Universal Robots URScript: motion_capture.script

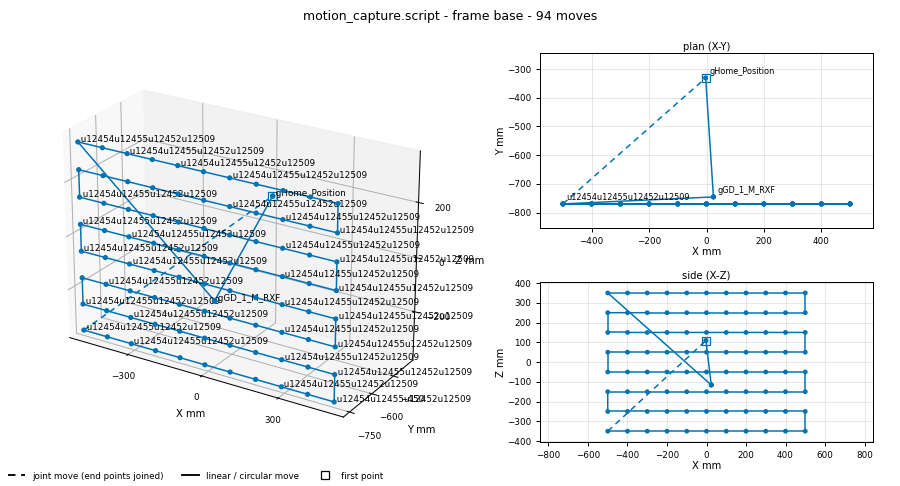
[picture p0: tool path of motion_capture.script in frame base, 94 of 94 moves have a stored position in this frame; points joined in program order, loops and branches not executed]
def motion_capture():
  global _hidden_verificationVariable=0
  set_standard_analog_input_domain(0, 1)
  set_standard_analog_input_domain(1, 1)
  set_tool_analog_input_domain(0, 1)
  set_tool_analog_input_domain(1, 1)
  set_analog_outputdomain(0, 0)
  set_analog_outputdomain(1, 0)
  set_input_actions_to_default()
  set_runstate_gp_boolean_output_to_value(0, 3)
  set_tcp(p[0.0,0.08,0.42,0.0,0.0,0.0])
  set_target_payload(0.100000, [0.135000, 0.000000, 0.225000], [10.000000, 10.000000, 10.000000, 0.000000, 0.000000, 0.000000])
  set_gravity([0.0, 0.0, 9.82])
  set_tool_communication(False, 115200, 0, 1, 1.5, 3.5)
  set_tool_output_mode(0)
  set_tool_digital_output_mode(0, 1)
  set_tool_digital_output_mode(1, 1)
  set_tool_voltage(0)
  set_safety_mode_transition_hardness(1)
  global DistPillar=0.26672
  global CandCnt=1
  global ReCaptZ=0.05
  global port=3000
  global socket_timeout=120
  global host="192.168.1.2"
  global is_popup=False
  global pBucket=[p[0.79266, 0.38712, 0.34284, 0, 0, -1.59403], p[-0.74859, -0.57465, 0.33542, 0, 0, 1.57589], p[0, 0, 0, 0, 0, 0]]
  global CaptStepZ=0.085
  global CaptIndex=[0, 0, 0]
  global pBucketM=p[-0.76064, -0.49997, 0.35503, 0, 0, 1.57135]
  global socket_name="vt"
  global rovi_err=0
  global SubPrgResult=100
  global CurrPos=p[-0.00509, -0.40914, 0.52153, -0.02622, -3.13819, -0.00861]
  global CurrPos_p=p[-0.00512, -0.32683, 0.10197, -0.02622, -3.13819, -0.00861]
  global ForceStartZ=0.4
  global CutOffZ=0.08
  global Sub3100_ZMax=0.74
  global ForceStartX=-0.90368
  global Sub3100_aRot=0.2
  global Sub3100_d=0.3
  global Sub3100_Option=3
  global Sub3100_a=0.2
  global Sub3100_XdV=0.1
  global Sub3100_XdRot=8
  global ZoneDistTh=0.05
  global BucketWidth=0.95
  global ZoneBucketGap=0
  global ZoneHomeX=0.2
  global UnloadZ=0.06
  global CaptPos=p[0.47573, -0.4259, 0.04497, 3.14138, 0.03448, 0.00005]
  global BucketUpperPos=p[0.47573, -0.4259, 0.04497, 3.14138, 0.03448, 0.00005]
  global Sub3100_GPII18=3
  global Zone6ThX=0.1
  global Zone6ThY=0.05
  global pCV=p[0.0013, 0.00002, 0.00241, 0.00218, 0.00027, 0.00056]
  global CaptRowNo=0
  global CrankDepthFull=0.025
  global CrankDepth=0.42751
  global Y1=[1, 266.72156, 0, 0]
  global Y2=p[0.01216, -0.30795, 0.04758, -0.01683, 0.01631, -1.59125]
  global EvacRadiusTh=0.3
  global EvacXTh=[-0.5, 0.5]
  global EvacYTh=[-0.8, 1]
  global EvacZTh=[-0.1, 0.1]
  global WorkPosNo=1
  global Zone1ZTh=0.1
  global ReCaptNo=0
  global DistPillarBak=0.26672
  global CaptIndexWk=0
  global PoseSub=p[-0.02953, -0.26506, -0.34451, -0.05387, -0.00646, 0.16446]
  global PoseAdd=p[-0.83785, 0.22711, 0.71052, 2.06849, 2.21352, 0.02519]
  global RZTh=15
  global pBucketC=p[0.45, -0.8, 0.35, 0, 0, 3.1415]
  global ReCaptZWk=0
  global CheckMST=2
  global RZSub=9.42295
  global DistPillarCOTh=0.16
  global DistPillarAPTh=0.25
  global CutOffZAdd=0.03
  global CutOffZDef=0.08
  global Y8=0
  global BKWidth_Value=[950, 986, 0]
  global BKWidth_Name="/prepro/bucket_width"
  global Bucket=p[0.32604,0.49174,0.0,-1.882900624652718E-5,2.8304179127934987E-5,-1.593185305749222]
  global BucketM=p[0.32604,0.49174,0.0,2.2353980716304163E-16,-3.5868426080024975E-16,-1.5931853071795856]
  global CV=p[0.0,0.0,0.0,0.0,0.0,0.0]
  global CaptPoint_C=p[-0.335,-0.024,0.4,-2.196299060524223,-2.2462891909035143,-5.664484063487096E-5]
  global CaptPoint_C2=p[0.32796661698047924,-0.010768520544682924,0.01931625281283378,2.2288103429550152,-2.213636886217198,8.598462540813273E-5]
  global CaptPoint_L=p[-0.335,-0.246,0.4,2.1515798175986935,2.2007172931471577,-0.09388261158531223]
  global CaptPoint_L2=p[0.327894307417917,-0.010799940826224014,0.01928712668893995,2.087717047309385,-2.0736781215133306,0.27365839887453103]
  global CaptPoint_R=p[-0.335,0.246,0.4,-2.1517289105627166,-2.2005994980169152,-0.09391633243318627]
  global CaptPoint_R2=p[0.327926308680866,-0.010795166414457658,0.019300245403843563,-2.1186306375223185,2.1040550557443427,0.22023197678473694]
  global Capt_1BK_L=p[-0.395,-0.47,0.35,-2.1961210242572884,-2.2463362846055,-2.908274762447041E-4]
  global Capt_1BK_R=p[-0.395,0.51,0.35,2.196067754706757,2.246288285862388,2.8411291050601595E-5]
  global Capt_1BK_pos1=p[-0.4218793038724447,-0.003154429464978058,0.2915499891144615,-2.1963422029204875,-2.2438663520270015,-0.02197160668673838]
  global Capt_1BK_pos2=p[-0.42187829024618434,-0.0031710253373066375,0.29156503858953065,-2.196324918349679,-2.2439040699490773,-0.021928444416953782]
  global Capt_2BK_L=p[0.42186661528427194,0.4254738068040517,0.35042275762909847,2.239156309475874,-2.1837044610999294,0.002643817066643282]
  global Capt_2BK_R=p[0.4218208572756906,-0.5427676723257963,0.350372239919558,2.2392697861179327,-2.183553596194912,0.002410470905346486]
  global Capt_2BK_pos1=p[0.42193501458435656,0.004742683868356356,0.35045865974037793,2.2391012408536453,-2.1839704655717003,0.002677867056024068]
  global Capt_2BK_pos2=p[0.421903984494575,0.004707988774967922,0.35045218900915065,2.239114367170047,-2.183895515396197,0.002684056681074047]
  global Capt_CV_M=p[-0.04794223960540197,-0.559868557160475,0.1086937653706071,-0.022464429848058916,-3.141454018347238,4.0166993855964835E-4]
  global Capt_GD_M=p[-0.004053197679954899,-0.25261725691632436,-0.01970497430780127,0.0332779454553888,-3.140179196376707,-0.0034093680964018282]
  global HomePointL=p[-0.36789,-0.5117344641471838,0.78,-0.6278857271586024,3.0680899128661667,-8.649957362498864E-4]
  global Master_pos=p[-0.003,-0.27,0.109,-0.02099899522131702,-3.141447277644474,4.6083856157132165E-4]
  global Master_posL=p[-0.003,-0.27,0.109,0.02094395102393583,3.0543261909900803,-5.235987755386035E-4]
  global Master_posR=p[-0.003,-0.27,0.109,-0.019810987664379186,-3.054193931591229,4.952746915529204E-4]
  global PickPos=p[0.10830682331105715,-1.3709505888096256,-0.18404188875951455,-0.00622194000158997,2.880236948927292,-0.00383636509397631]
  global Solve=p[-0.00368,-0.0021000000000000003,0.25739999999999996,0.0,0.0,0.0]
  global TCP3100TL=p[0.0,0.06,0.535,1.8939999999999997,0.0,0.0]
  global TEST=p[0.1,0.0,0.2,0.0,0.0,0.0]
  global UF=p[0.0,0.0,0.0,0.0,0.0,0.0]
  global g1CV_posL1=p[0.05028133628211688,-0.4526481033729615,0.1221845548632916,-2.213335080948508,-2.1937561336067057,-0.3280056759040735]
  global g1CV_posR1=p[0.03743870476062511,-0.53119407812668,0.11301901343688614,2.073418671558482,2.153257467049566,0.11656306439039889]
  global g1GD_pos1=p[0.14857012745627257,-0.6379982996093139,0.2691918735517042,2.214277610229479,2.228493098198348,-1.6896832945346036E-4]
  global g1GD_pos2=p[0.028634297882679793,-0.4702313285867709,0.450031657325677,2.214319081558633,2.2285182736309666,-1.5473710223511705E-5]
  global g1GD_pos3=p[-0.1945307709581842,-0.42906455111749103,0.45,-2.685709191057467,-1.6297557787554324,7.112239955701245E-5]
  global g1GD_pos4=p[-0.25628841794770224,-0.020630481098425146,0.45,2.148716725221303,2.2918109407224354,-1.3854918368741778E-5]
  global g1GD_pos5=p[-0.714365317693782,-0.022971007293656684,0.45,-2.1476725881724037,-2.292771958266831,6.311233907547867E-5]
  global g1GD_posL1=p[-0.08276848269606216,-0.3996147100031649,0.1488453551331823,2.286527078917204,1.8420745504477611,0.33698451773695576]
  global g1GD_posL2=p[-0.3253977027403738,-0.3024804624281039,0.16332814085945146,2.72312820760317,0.9631021078169197,0.32447452035226126]
  global g1GD_posL3=p[-0.6791033397183219,0.06787475590683856,0.16337212788108813,2.1383125299263996,2.086116032377724,0.4536080263755059]
  global g1GD_posR1=p[-0.09893370538053747,-0.4999608954567234,0.14329885217724153,2.43311852414254,1.4238397520832589,0.08559216753941556]
  global g1GD_posR2=p[-0.3729565201882258,-0.3752983669473301,0.143299052800563,2.6951655216297596,0.8130506811102118,-0.02387549506099888]
  global g1GD_posR3=p[-0.7385929502572233,-0.029472684480355026,0.1499650660949685,2.0484522752014467,1.9493695704119496,0.18368227556562683]
  global g2CV_posL1=p[0.3409386496330911,-0.4656338066361442,0.1250074988128972,2.209372209162659,2.1945371304665926,0.3160714960040194]
  global g2CV_posR1=p[0.3400736278759575,-0.531334269888987,0.1183415684753657,2.07314649492589,2.1532617466521136,0.11638666128062146]
  global g2GD_pos1=p[0.2541383831722086,-0.6774928758666339,0.18519960582577166,-2.0375719953016755,-2.3889847960447277,-0.0020926217702447064]
  global g2GD_pos2=p[0.2548303032832998,-0.4395886120507379,0.2986557393825452,-1.8691601740155521,-2.5210138137905886,-0.00387894312889377]
  global g2GD_pos3=p[0.3379879014596998,-0.06467509721500111,0.3,-0.13681955358471554,3.138134920213652,0.0052602971824959885]
  global g2GD_pos4=p[0.31412137931928874,0.14047894136547145,0.3,1.0726627132331576,-2.952135651121033,-0.005044331815994264]
  global g2GD_pos5=p[0.596826867485263,0.012800854207951809,0.3,-2.250960447020382,2.191482163995288,-8.62049956035814E-5]
  global gCV_11_M=p[0.2895856132087369,-0.9700402997477822,-0.03048660701646616,2.1152349881492576,2.082454134650371,0.2907202126305862]
  global gCV_12_M=p[0.3399735651774522,-0.9701152791174454,-0.030398240983259495,2.1151309943729695,2.082422893849917,0.2905107745619789]
  global gCV_13_M=p[0.3677028242565019,-0.8912043588518235,0.06406475497489328,2.0725171273330782,1.9964853271438565,0.36457536397978224]
  global gCV_1_M=p[0.26662,-0.9702099878169796,-0.021959001781271192,-2.212353529315613,-2.2195544467592487,0.0323655800559973]
  global gCV_2_M=p[0.26859807289598814,-0.9702702137427199,0.029436000792852024,-2.212446744366122,-2.219572570655569,0.03244046687031327]
  global gCV_3_M=p[0.29099390607376485,-0.6570558385379063,0.0722153583041818,1.9884242634571576,2.2321538498123994,0.15249643504377583]
  global gCV_pos5=p[0.3400172856834047,-0.9722754606605235,-0.18287928563575456,2.073394561413637,2.1531827558666565,0.11639000988241816]
  global gGD_1_LM=p[0.02419,-0.7289500000000001,-0.11494,-0.010169347158913017,2.870767181856166,0.2884627079222753]
  global gGD_1_LM_RX=p[0.05369459866460638,-0.7259829268100212,-0.22783950231933825,0.3045827799067659,1.9676452376021116,-2.225919618395937]
  global gGD_1_LM_RXF=p[0.02413503458160308,-0.74534,-0.11578000000000001,0.2411332216392182,1.7407173006243832,-2.3674279033231747]
  global gGD_1_M=p[0.023469999999999998,-0.72661,-0.11456000000000001,-0.029570847824802682,-3.12419917405015,-0.3106340785404749]
  global gGD_1_M_RX=p[0.023057660296999655,-0.7236214973426132,-0.23125683282505294,-0.014877844076808725,-2.067340942848176,2.343588104915257]
  global gGD_1_M_RXF=p[0.02415523713330076,-0.7453200000000001,-0.11578426509069895,-0.012477314995716382,-1.853515977408631,2.515027308648709]
  global gGD_1_RM=p[0.023629999999999998,-0.72653,-0.11331000000000001,-0.06253229749015264,-2.8808212567082414,-0.28238046714011755]
  global gGD_1_RM_RX=p[-0.005088870384171898,-0.7236679006721032,-0.22637303238730694,0.2593876111855818,-1.9494145656951658,2.2163695295960366]
  global gGD_1_RM_RXF=p[0.024158234647744328,-0.74536,-0.11577,0.21548497967238725,-1.726437707763004,2.3373117534316665]
  global gGD_2_LM=p[0.02467,-0.67055,-0.11509,-0.010179461791212513,2.870955921048522,0.2878734195391217]
  global gGD_2_LM_RX=p[0.05420311073735988,-0.6676020823088724,-0.22799649297520497,0.30453821192036695,1.967284185886619,-2.2263172758170806]
  global gGD_2_LM_RXF=p[0.02518,-0.6822999999999999,-0.11982,0.24121310672797797,1.7407223643292684,-2.3672997334921986]
  global gGD_2_M=p[0.02389,-0.6721900000000001,-0.11456000000000001,-0.029666521928107308,-3.1243201149134068,-0.3098990972493868]
  global gGD_2_M_RX=p[0.023451397096722927,-0.6694131949440525,-0.2312112380080017,-0.014956274784115499,-2.0665404158707275,2.344308336230428]
  global gGD_2_M_RXF=p[0.02469,-0.68228,-0.11781,-0.012625584579695818,-1.8536977166603092,2.514979910589354]
  global gGD_2_RM=p[0.02429,-0.66916,-0.11353,-0.06253008389277029,-2.880917079483223,-0.28230802316028863]
  global gGD_2_RM_RX=p[-0.004446905642647561,-0.6662749600062835,-0.22659916730049184,0.25917451838034067,-1.9493834256574814,2.2163998591438716]
  global gGD_2_RM_RXF=p[0.02418,-0.68221,-0.11985,0.21545635593876583,-1.7267658137434814,2.337110041109278]
  global gGD_3_LM=p[0.024149999999999998,-0.63442,-0.00372,-0.010168641563882792,2.8709293839329573,0.28786844960240987]
  global gGD_3_LM_RX=p[0.05363363651684515,-0.6315154925298007,-0.11660858214565634,0.3044658366193896,1.9671814668034862,-2.2263956155853166]
  global gGD_3_LM_RXF=p[0.02387752228160463,-0.5964211774687285,-0.05792315514989682,0.2704410553277331,1.9481847980902196,-2.214876983085744]
  global gGD_3_M=p[0.023940000000000003,-0.63613,-0.00522,-0.029962916255114207,-3.1241595671421933,-0.3100480455299553]
  global gGD_3_M_RX=p[0.023480543069899083,-0.6332104768802226,-0.1219058093136538,-0.014942206094503903,-2.066644773324154,2.3438407418712903]
  global gGD_3_M_RXF=p[0.02383447419609676,-0.5964085561522618,-0.0579509198373786,-0.014600929068906539,-2.066655165579624,2.3438719244209403]
  global gGD_3_RM=p[0.02428,-0.6347200000000001,-0.00846,-0.0624152449577923,-2.8809080008278345,-0.2823877130468296]
  global gGD_3_RM_RX=p[-0.004516944470436435,-0.6317425605459723,-0.12157603214553458,0.2593921862362061,-1.9496410574300858,2.2162312511396824]
  global gGD_3_RM_RXF=p[0.023773322279514588,-0.5964087734876792,-0.05795139315103717,0.24060086319727583,-1.933030903056379,2.187075285864524]
  global gGD_4_LM=p[-0.12534109989305553,-0.6345452257364079,-0.003660409912739915,-0.010209507081901941,2.87092276677584,0.2878514545752189]
  global gGD_4_RM=p[0.1741356102640685,-0.6348673415405857,-0.008407071546374267,-0.06250935255312234,-2.8810578033032743,-0.28204363282303685]
  global gHome_Position=p[-0.0028799999999999997,-0.33081,0.1087,-0.02099958342773921,-3.141491282453575,3.986162810876369E-4]
  global gTAIHI_pos1=p[0.034435296708333146,-0.2890869270984411,0.28697762766096685,-0.9517096680276043,2.9907327255336362,-0.006242657270483182]
  global gTAIHI_pos2=p[0.46041690381401934,0.09562026346103787,0.3409455343940188,-2.575428180750575,1.7504967205574518,-0.009370784990557466]
  global gTAIHI_pos3=p[0.4777514786587304,0.10855417509450788,0.25667938190447326,-3.115092130529677,-0.059113053813058626,0.017060902648732133]
  global gTAIHI_pos4=p[0.47773948064032057,0.10853581553326999,-0.15133852019421468,-3.1151611852917296,-0.05914313994407087,0.017149581050184888]
  global gTAIHI_pos5=p[0.30588450070104545,0.17870028478253597,-0.38750721344025674,-3.115302721311487,-0.05927431563397507,0.01725874757592571]
  rtde_set_watchdog("speed_slider_mask", 10.0, "ignore")
  # begin: URCap Installation Node
  #   Source: Ethernet/IP I/O Monitor URCap, 1.0.0,
  #   Type: Ethernet/IP I/O Monitor
  conn = rpc_factory("xmlrpc", "http://127.0.0.1:" + to_str(61101) + "/RPC2")

  def show_monitor():
    return conn.eip_monitor.show()
  end
  # end: URCap Installation Node
  step_count_397ec1da_4bf5_4cd9_852d_7e56d1a44991 = 0.0
  thread Step_Counter_Thread_d30562aa_f9e6_4b1c_b905_026c51a4cdd0():
    while (True):
      step_count_397ec1da_4bf5_4cd9_852d_7e56d1a44991 = step_count_397ec1da_4bf5_4cd9_852d_7e56d1a44991 + 1.0
      sync()
    end
  end
  run Step_Counter_Thread_d30562aa_f9e6_4b1c_b905_026c51a4cdd0()
  global u12454u12455u12452u12509u12452u12531u12488_1_p=p[-.500000000000, -.769756443525, .350000000000, .026412316980, 3.122703155576, .190069130431]
  global u12454u12455u12452u12509u12452u12531u12488_1_q=[-1.9114113979977487, -2.2618906676528763, -0.4591602097308458, -2.1103464893291033, 1.5382040123912875, -0.3218736006056453]
  global u12454u12455u12452u12509u12452u12531u12488_2_p=p[-.400000000000, -.769779294180, .350000000000, .026483300731, 3.122677399875, .189931430077]
  global u12454u12455u12452u12509u12452u12531u12488_2_q=[-1.8171775039295675, -2.133570399697568, -0.6739164307743053, -2.0258656041570973, 1.5500367362507816, -0.22781589719288586]
  global u12454u12455u12452u12509u12452u12531u12488_3_p=p[-.300000000000, -.769789509042, .350000000000, .026503166818, 3.122680364614, .190021042089]
  global u12454u12455u12452u12509u12452u12531u12488_3_q=[-1.716165423221513, -2.0483178045096206, -0.8067403790800718, -1.9793255819153632, 1.5626303580459329, -0.12725853176687707]
  global u12454u12455u12452u12509u12452u12531u12488_4_p=p[-.200000000000, -.769710320339, .350000000000, .026644809517, 3.122684897999, .190163528053]
  global u12454u12455u12452u12509u12452u12531u12488_4_q=[-1.6099254452403873, -1.9903140904082264, -0.8928752732962089, -1.9509751362852477, 1.5758064426187728, -0.021545386634477026]
  global u12454u12455u12452u12509u12452u12531u12488_5_p=p[-.100000000000, -.769748949148, .350000000000, .026539604733, 3.122630476655, .190199683938]
  global u12454u12455u12452u12509u12452u12531u12488_5_q=[-1.5005112395057907, -1.9556374381444463, -0.9429912511335443, -1.9338143920604765, 1.5892342589142574, 0.08710325076008775]
  global u12454u12455u12452u12509u12452u12531u12488_6_p=p[-.000000000000, -.769753039159, .350000000000, .026417422847, 3.122605840141, .190062143068]
  global u12454u12455u12452u12509u12452u12531u12488_6_q=[-1.3903873476760396, -1.9425809473745055, -0.9620710317474312, -1.924501091481389, 1.6023466178665648, 0.19644588241672967]
  global u12454u12455u12452u12509u12452u12531u12488_7_p=p[.100000000000, -.769697827339, .350000000000, .026676373995, 3.122609886009, .190250248267]
  global u12454u12455u12452u12509u12452u12531u12488_7_q=[-1.2822308148508128, -1.951096029905166, -0.9510725611357058, -1.9225876310592298, 1.6147201968064984, 0.3041064480521222]
  global u12454u12455u12452u12509u12452u12531u12488_8_p=p[.200000000000, -.769720790847, .350000000000, .026556961083, 3.122644596660, .190093490077]
  global u12454u12455u12452u12509u12452u12531u12488_8_q=[-1.17843186168205, -1.9812086634530637, -0.9092976431058046, -1.9286067868835772, 1.6258983197269878, 0.4072497591845611]
  global u12454u12455u12452u12509u12452u12531u12488_9_p=p[.300000000000, -.769733702676, .350000000000, .026566917094, 3.122644604456, .190111967042]
  global u12454u12455u12452u12509u12452u12531u12488_9_q=[-1.0809947819676138, -2.0340650931016366, -0.832913028063154, -1.9458910758426562, 1.6357754765791155, 0.5041839537901349]
  global u12454u12455u12452u12509u12452u12531u12488_10_p=p[.400000000000, -.769744499214, .350000000000, .026575326306, 3.122733131353, .190132184073]
  global u12454u12455u12452u12509u12452u12531u12488_10_q=[-0.991056047875758, -2.112822831401303, -0.7130015422450269, -1.9804884405124454, 1.6441329192153846, 0.5936653453753264]
  global u12454u12455u12452u12509u12452u12531u12488_11_p=p[.500000000000, -.769782793267, .350000000000, .026508483411, 3.122675353931, .190004333780]
  global u12454u12455u12452u12509u12452u12531u12488_11_q=[-0.9092045285356001, -2.2282728608507227, -0.5245252474117779, -2.0467514170930947, 1.6511301529893736, 0.674987056963054]
  global u12454u12455u12452u12509u12452u12531u12488_12_p=p[.500000000000, -.769760900368, .250000000000, .026528118536, 3.122708730810, .190029220965]
  global u12454u12455u12452u12509u12452u12531u12488_12_q=[-0.91001526414599, -2.1575818481165623, -0.8234281729531467, -1.8186342475237138, 1.6514532038321557, 0.674277213721763]
  global u12454u12455u12452u12509u12452u12531u12488_13_p=p[.400000000000, -.769733463067, .250000000000, .026514979020, 3.122645894238, .190244682604]
  global u12454u12455u12452u12509u12452u12531u12488_13_q=[-0.9917864872644486, -2.066558737990783, -0.9638838946787551, -1.775946946298058, 1.6445187709217466, 0.5928948733369976]
  global u12454u12455u12452u12509u12452u12531u12488_14_p=p[.300000000000, -.769779850713, .250000000000, .026486137196, 3.122687044148, .190087115632]
  global u12454u12455u12452u12509u12452u12531u12488_14_q=[-1.0815959341128414, -1.9988992643907082, -1.0626874450643164, -1.7513322373267535, 1.6359840099262097, 0.5034994136646239]
  global u12454u12455u12452u12509u12452u12531u12488_15_p=p[.200000000000, -.769781810740, .250000000000, .026484014283, 3.122705057460, .190154645546]
  global u12454u12455u12452u12509u12452u12531u12488_15_q=[-1.178993777620991, -1.9517406172159042, -1.1285374498245746, -1.7389315215400138, 1.6260890541146251, 0.4065892996566263]
  global u12454u12455u12452u12509u12452u12531u12488_16_p=p[.100000000000, -.769767054232, .250000000000, .026526291040, 3.122613308500, .190027323171]
  global u12454u12455u12452u12509u12452u12531u12488_16_q=[-1.2827714411646953, -1.9240889198247118, -1.165721384028017, -1.7348376877857614, 1.614912560975787, 0.3034134866458757]
  global u12454u12455u12452u12509u12452u12531u12488_17_p=p[-.000000000000, -.769774212018, .250000000000, .026548873992, 3.122655101521, .190254700093]
  global u12454u12455u12452u12509u12452u12531u12488_17_q=[-1.3909214332126858, -1.9163049894413131, -1.1754366000499896, -1.737561855870414, 1.6025377303774226, 0.19593182526004416]
  global u12454u12455u12452u12509u12452u12531u12488_18_p=p[-.100000000000, -.769761106494, .250000000000, .026526373802, 3.122686049502, .190157333824]
  global u12454u12455u12452u12509u12452u12531u12488_18_q=[-1.501031671994486, -1.9279015874596954, -1.1588712635165734, -1.7456586341412317, 1.5894077694755506, 0.08651688314535733]
  global u12454u12455u12452u12509u12452u12531u12488_19_p=p[-.200000000000, -.769774136564, .250000000000, .026456934430, 3.122604840588, .190033566826]
  global u12454u12455u12452u12509u12452u12531u12488_19_q=[-1.6105390632010685, -1.9591661196706518, -1.1149754495250734, -1.759952863358695, 1.5761181644969744, -0.02233440855401625]
  global u12454u12455u12452u12509u12452u12531u12488_20_p=p[-.300000000000, -.769781720580, .250000000000, .026577890837, 3.122652970758, .190179047147]
  global u12454u12455u12452u12509u12452u12531u12488_20_q=[-1.7167999596103485, -2.010364020103964, -1.0415152543063009, -1.7826055876402425, 1.5628826553775266, -0.12787467040920664]
  global u12454u12455u12452u12509u12452u12531u12488_21_p=p[-.400000000000, -.769744400680, .250004230661, .026455713576, 3.122633726963, .190216871674]
  global u12454u12455u12452u12509u12452u12531u12488_21_q=[-1.8178876271517623, -2.0823453079114493, -0.9341277490262669, -1.8170533568045393, 1.5502952050585215, -0.22852714499667925]
  global u12454u12455u12452u12509u12452u12531u12488_22_p=p[-.500000000000, -.769752806148, .249977272123, .026544126851, 3.122621458039, .190284973089]
  global u12454u12455u12452u12509u12452u12531u12488_22_q=[-1.912334332224173, -2.179253324474807, -0.7817836665202043, -1.870495209636136, 1.53856375120108, -0.32259002476777]
  global u12454u12455u12452u12509u12452u12531u12488_23_p=p[-.500000000000, -.769728484770, .150000000000, .026393123076, 3.122651774268, .190178886745]
  global u12454u12455u12452u12509u12452u12531u12488_23_q=[-1.9128442312041365, -2.1609661241967473, -0.987071729191296, -1.683405002467147, 1.538744683268341, -0.32326048625640524]
  global u12454u12455u12452u12509u12452u12531u12488_24_p=p[-.400000000000, -.769776260329, .150000000000, .026496921071, 3.122616212816, .190058872149]
  global u12454u12455u12452u12509u12452u12531u12488_24_q=[-1.8183484767892821, -2.0756758619090068, -1.119625076860153, -1.638125740464143, 1.5504998869009539, -0.2290611172505086]
  global u12454u12455u12452u12509u12452u12531u12488_25_p=p[-.300000000000, -.769742523564, .149972007931, .026671481565, 3.122589595262, .190100603900]
  global u12454u12455u12452u12509u12452u12531u12488_25_q=[-1.7172499604707783, -2.0100622561114037, -1.217213616444221, -1.6071690471086697, 1.5630915763257234, -0.1283793186395803]
  global u12454u12455u12452u12509u12452u12531u12488_26_p=p[-.200000000000, -.769780338502, .149978041748, .026528023660, 3.122636425681, .190070149226]
  global u12454u12455u12452u12509u12452u12531u12488_26_q=[-1.610892382818097, -1.9627414022092786, -1.2852160392852294, -1.5861622342848385, 1.5762157500238576, -0.02275843600603178]
  global u12454u12455u12452u12509u12452u12531u12488_27_p=p[-.100000000000, -.769745881180, .149995549479, .026451519491, 3.122618883192, .190101837112]
  global u12454u12455u12452u12509u12452u12531u12488_27_q=[-1.5014170801735727, -1.9334650534417097, -1.3264985118771904, -1.5724417136414282, 1.5895919353511783, 0.08595968623292746]
  global u12454u12455u12452u12509u12452u12531u12488_28_p=p[.000000000000, -.769794456996, .149992141995, .026554396761, 3.122606353239, .190010846636]
  global u12454u12455u12452u12509u12452u12531u12488_28_q=[-1.3912924404706617, -1.9226155501285076, -1.3421332945507913, -1.5644092481035372, 1.6026905136881453, 0.19544350978913963]
  global u12454u12455u12452u12509u12452u12531u12488_29_p=p[.100000000000, -.769806987713, .149985740336, .026560443917, 3.122586219799, .189931438497]
  global u12454u12455u12452u12509u12452u12531u12488_29_q=[-1.2831438437635398, -1.9302091184868697, -1.332632629894107, -1.5617624067960563, 1.6150494824601616, 0.3029425526560603]
  global u12454u12455u12452u12509u12452u12531u12488_30_p=p[.200000000000, -.769814423607, .150010855459, .026516643396, 3.122584097137, .189982361164]
  global u12454u12455u12452u12509u12452u12531u12488_30_q=[-1.1794180535327925, -1.956237208193265, -1.2974749489939068, -1.5653811410892091, 1.6262953338083186, 0.40606816526849876]
  global u12454u12455u12452u12509u12452u12531u12488_31_p=p[.300000000000, -.769831553064, .150060942487, .026545222581, 3.122662417995, .189866103692]
  global u12454u12455u12452u12509u12452u12531u12488_31_q=[-1.0819925902355525, -2.0002866059266946, -1.2357744304054723, -1.576750564863108, 1.6360955536829191, 0.5030348882059403]
  global u12454u12455u12452u12509u12452u12531u12488_32_p=p[.400000000000, -.769795781366, .150028602698, .026503365861, 3.122587531329, .189968750155]
  global u12454u12455u12452u12509u12452u12531u12488_32_q=[-0.9922270738397705, -2.0624181412994282, -1.1453333100908685, -1.5984937767840375, 1.6446469758576996, 0.5923566878529133]
  global u12454u12455u12452u12509u12452u12531u12488_33_p=p[.500000000000, -.769793999499, .150020314544, .026447218837, 3.122575290255, .189986171446]
  global u12454u12455u12452u12509u12452u12531u12488_33_q=[-0.9105654759643107, -2.1436878918100923, -1.0211433188916939, -1.634766430642408, 1.6517313132940015, 0.6736049555830492]
  global u12454u12455u12452u12509u12452u12531u12488_34_p=p[.500000000000, -.769779861568, .050000000000, .026542041208, 3.122557555389, .190062616528]
  global u12454u12455u12452u12509u12452u12531u12488_34_q=[-0.9108895793250085, -2.1632011203124684, -1.1662261267105478, -1.4702404330490406, 1.6518725992844814, 0.6731792662005232]
  global u12454u12455u12452u12509u12452u12531u12488_35_p=p[.400000000000, -.769760513107, .050000000000, .026549866540, 3.122587439777, .190000613354]
  global u12454u12455u12452u12509u12452u12531u12488_35_q=[-0.9924845968610327, -2.0881935330063115, -1.2831795311436416, -1.4349224479921512, 1.6447338235902051, 0.5919582930454563]
  global u12454u12455u12452u12509u12452u12531u12488_36_p=p[.300000000000, -.769793437396, .050000000000, .026367160197, 3.122672293278, .190001319070]
  global u12454u12455u12452u12509u12452u12531u12488_36_q=[-1.0822201887748832, -2.0301660421005394, -1.3699155602403739, -1.4128452711626203, 1.636174279208616, 0.5025162468030526]
  global u12454u12455u12452u12509u12452u12531u12488_37_p=p[.200000000000, -.769726213919, .050000000000, .026627232633, 3.122697997976, .190137353324]
  global u12454u12455u12452u12509u12452u12531u12488_37_q=[-1.1795709628866948, -1.9885443352899195, -1.4298833078132702, -1.4008180335198368, 1.6262735945297104, 0.40581240128416063]
  global u12454u12455u12452u12509u12452u12531u12488_38_p=p[.100000000000, -.769733672147, .050000000000, .026554565165, 3.122685196493, .190232809370]
  global u12454u12455u12452u12509u12452u12531u12488_38_q=[-1.283303317577559, -1.963915417659761, -1.4641828291134331, -1.3967363080991797, 1.6150349457186142, 0.3026044310190157]
  global u12454u12455u12452u12509u12452u12531u12488_39_p=p[.000000000000, -.769785322216, .050000000000, .026510503638, 3.122723125005, .190004512455]
  global u12454u12455u12452u12509u12452u12531u12488_39_q=[-1.3914339238266074, -1.9565180079824351, -1.4737422544074672, -1.3989224808881673, 1.6026155458683435, 0.1951072590510945]
  global u12454u12455u12452u12509u12452u12531u12488_40_p=p[-.100000000000, -.769765413659, .050000000000, .026427054269, 3.122646229983, .190092806256]
  global u12454u12455u12452u12509u12452u12531u12488_40_q=[-1.5016202252969766, -1.9667091354205404, -1.458514209701086, -1.407185734712944, 1.5896005709127916, 0.0855699677390378]
  global u12454u12455u12452u12509u12452u12531u12488_41_p=p[-.200000000000, -.769712657217, .050000000000, .026669437619, 3.122668765801, .190172396507]
  global u12454u12455u12452u12509u12452u12531u12488_41_q=[-1.6111137968452418, -1.9941576858132901, -1.4184742805621404, -1.4215535025581794, 1.5762220127117197, -0.023059579298967847]
  global u12454u12455u12452u12509u12452u12531u12488_42_p=p[-.300000000000, -.769708675215, .050000000000, .026592329375, 3.122688586472, .190100650432]
  global u12454u12455u12452u12509u12452u12531u12488_42_q=[-1.717446082348145, -2.038485220608205, -1.3528387367862003, -1.443102243336619, 1.563050842151673, -0.1287922067915055]
  global u12454u12455u12452u12509u12452u12531u12488_43_p=p[-.400000000000, -.769723587764, .050000000000, .026548087776, 3.122655882932, .190070701895]
  global u12454u12455u12452u12509u12452u12531u12488_43_q=[-1.8186227366851835, -2.099509098658128, -1.259828810329843, -1.4740780696228883, 1.5505307857911361, -0.22946732186074925]
  global u12454u12455u12452u12509u12452u12531u12488_44_p=p[-.500000000000, -.769745444991, .050000000000, .026448305973, 3.122671770036, .190070038317]
  global u12454u12455u12452u12509u12452u12531u12488_44_q=[-1.913168549752596, -2.1777485306121296, -1.1359749765764775, -1.5176355928160845, 1.5388491761007717, -0.3237064384801265]
  global u12454u12455u12452u12509u12452u12531u12488_45_p=p[-.500000000000, -.769748044989, -.050000000000, .026459265213, 3.122632683617, .190122460314]
  global u12454u12455u12452u12509u12452u12531u12488_45_q=[-1.9133780773117284, -2.2211331388335616, -1.2450197950729933, -1.3652385838548202, 1.5388943999966873, -0.32413817674840395]
  global u12454u12455u12452u12509u12452u12531u12488_46_p=p[-.400000000000, -.769739650303, -.050000000000, .026524363418, 3.122756240847, .190055765096]
  global u12454u12455u12452u12509u12452u12531u12488_46_q=[-1.8187371277192126, -2.1486524407136685, -1.3647457810366612, -1.3199753277104946, 1.5504419407841503, -0.22982482924301184]
  global u12454u12455u12452u12509u12452u12531u12488_47_p=p[-.300000000000, -.769776202108, -.050000000000, .026395617042, 3.122681115272, .190056900613]
  global u12454u12455u12452u12509u12452u12531u12488_47_q=[-1.7175787153903785, -2.091961769853695, -1.4555700035182593, -1.286866813305382, 1.5630389047729167, -0.1292835164360282]
  global u12454u12455u12452u12509u12452u12531u12488_48_p=p[-.200000000000, -.769746729862, -.050000000000, .026524482261, 3.122666596847, .190157077818]
  global u12454u12455u12452u12509u12452u12531u12488_48_q=[-1.6112382773031273, -2.050586009680634, -1.5203481415147833, -1.263245226402418, 1.5761868010532227, -0.023506832417726997]
  global u12454u12455u12452u12509u12452u12531u12488_49_p=p[-.100000000000, -.769781536209, -.050000000000, .026509312290, 3.122634166369, .189996544206]
  global u12454u12455u12452u12509u12452u12531u12488_49_q=[-1.5017608226441368, -2.0249283672268668, -1.5600934719950121, -1.2473325509067834, 1.589570965909667, 0.08525364952997627]
  global u12454u12455u12452u12509u12452u12531u12488_50_p=p[-.000000000000, -.769750846669, -.050000000000, .026510672437, 3.122715317755, .189959048159]
  global u12454u12455u12452u12509u12452u12531u12488_50_q=[-1.3915520266447254, -2.0154486486529937, -1.5752093407577448, -1.2385065815255096, 1.6025755644109516, 0.19476181077474664]
  global u12454u12455u12452u12509u12452u12531u12488_51_p=p[.100000000000, -.769758377488, -.050000000000, .026415226178, 3.122608928546, .189993842825]
  global u12454u12455u12452u12509u12452u12531u12488_51_q=[-1.2834508712456465, -2.022498172237963, -1.5655654952664868, -1.2366210119909358, 1.6150294159800644, 0.30214056754365615]
  global u12454u12455u12452u12509u12452u12531u12488_52_p=p[.200000000000, -.769741232078, -.050000000000, .026477631813, 3.122639493213, .190040124831]
  global u12454u12455u12452u12509u12452u12531u12488_52_q=[-1.1797194426026554, -2.0457471515932006, -1.5312483524744307, -1.2421947195565437, 1.6262708325806638, 0.40533732068220546]
  global u12454u12455u12452u12509u12452u12531u12488_53_p=p[.300000000000, -.769771253385, -.050000000000, .026440740859, 3.122680746441, .190105575992]
  global u12454u12455u12452u12509u12452u12531u12488_53_q=[-1.082367864250675, -2.0848313740485054, -1.47171795245423, -1.256467760367169, 1.636176291718435, 0.5021782940431911]
  global u12454u12455u12452u12509u12452u12531u12488_54_p=p[.400000000000, -.769796136968, -.050000000000, .026521578517, 3.122636413280, .189965006196]
  global u12454u12455u12452u12509u12452u12531u12488_54_q=[-0.992637251316915, -2.139060043269442, -1.3864212946893275, -1.280849891309007, 1.6446845014586442, 0.5915537482108344]
  global u12454u12455u12452u12509u12452u12531u12488_55_p=p[.500000000000, -.769786059723, -.050000000000, .026316709790, 3.122664812943, .189943043569]
  global u12454u12455u12452u12509u12452u12531u12488_55_q=[-0.9110046564723726, -2.2086729582625964, -1.272963212183594, -1.3180640413277303, 1.6517761398124051, 0.6726918965713659]
  global u12454u12455u12452u12509u12452u12531u12488_56_p=p[.500000000000, -.769750842608, -.150000000000, .026576178818, 3.122698301473, .190011515803]
  global u12454u12455u12452u12509u12452u12531u12488_56_q=[-0.9110970984109397, -2.276252383856396, -1.347153303793216, -1.1763787854940624, 1.651757782315294, 0.6724576316309739]
  global u12454u12455u12452u12509u12452u12531u12488_57_p=p[.400000000000, -.769754420921, -.150000000000, .026432926505, 3.122687908541, .190236060830]
  global u12454u12455u12452u12509u12452u12531u12488_57_q=[-0.9927130052839024, -2.2120268892728383, -1.4589411504396814, -1.1355746884560123, 1.644668798620852, 0.5911068844867899]
  global u12454u12455u12452u12509u12452u12531u12488_58_p=p[.300000000000, -.769727558898, -.150000000000, .026443041315, 3.122710365311, .190070280384]
  global u12454u12455u12452u12509u12452u12531u12488_58_q=[-1.0823974304715982, -2.161768249631587, -1.5440824922106886, -1.107180888665253, 1.6360684770429463, 0.501849331153567]
  global u12454u12455u12452u12509u12452u12531u12488_59_p=p[.200000000000, -.769735598305, -.150000000000, .026509885840, 3.122665580848, .190106171381]
  global u12454u12455u12452u12509u12452u12531u12488_59_q=[-1.1797732273589716, -2.125771589194901, -1.6035225543618727, -1.0899655718696195, 1.626165111307913, 0.4050038772467283]
  global u12454u12455u12452u12509u12452u12531u12488_60_p=p[.100000000000, -.769718614799, -.150000000000, .026529489015, 3.122709660842, .190009796657]
  global u12454u12455u12452u12509u12452u12531u12488_60_q=[-1.2834457784971702, -2.1041965409259493, -1.6381762791250116, -1.082359179521898, 1.614837263632402, 0.30192630527617503]
  global u12454u12455u12452u12509u12452u12531u12488_61_p=p[.000000000000, -.769760786810, -.150000000000, .026491073828, 3.122659235698, .190092594337]
  global u12454u12455u12452u12509u12452u12531u12488_61_q=[-1.391643409580758, -2.0977128601711366, -1.6478043137865956, -1.0837378618532156, 1.6025222306578943, 0.19435870344199863]
  global u12454u12455u12452u12509u12452u12531u12488_62_p=p[-.100000000000, -.769767516941, -.150000000000, .026535738072, 3.122732471726, .189923741876]
  global u12454u12455u12452u12509u12452u12531u12488_62_q=[-1.5017615545766096, -2.10615090464895, -1.6329902605422326, -1.093176220192678, 1.5893735063179861, 0.08498044138937318]
  global u12454u12455u12452u12509u12452u12531u12488_63_p=p[-.200000000000, -.769762168209, -.150000000000, .026556031592, 3.122733063322, .189954225080]
  global u12454u12455u12452u12509u12452u12531u12488_63_q=[-1.6112753022876936, -2.1296173376021956, -1.5933212722006544, -1.1111095188625022, 1.5760440022231437, -0.023817333468188373]
  global u12454u12455u12452u12509u12452u12531u12488_64_p=p[-.300000000000, -.769777524075, -.150000000000, .026513705096, 3.122643188370, .189999118835]
  global u12454u12455u12452u12509u12452u12531u12488_64_q=[-1.7176873889359028, -2.167709033536277, -1.5286534696472849, -1.138004583086591, 1.56300417768342, -0.1296182406891031]
  global u12454u12455u12452u12509u12452u12531u12488_65_p=p[-.400000000000, -.769718014728, -.150000000000, .026599020811, 3.122672585016, .190075501102]
  global u12454u12455u12452u12509u12452u12531u12488_65_q=[-1.818878376231555, -2.2199564837641024, -1.4385857523532577, -1.1748586285275326, 1.5504577149311596, -0.2302227785129496]
  global u12454u12455u12452u12509u12452u12531u12488_66_p=p[-.500000000000, -.769744739345, -.150000000000, .026603673243, 3.122619884666, .190095930256]
  global u12454u12455u12452u12509u12452u12531u12488_66_q=[-1.9135073014201085, -2.2868035947719707, -1.3208854648621937, -1.2236800329525934, 1.5388881729639545, -0.32447693995867066]
  global u12454u12455u12452u12509u12452u12531u12488_67_p=p[-.500002619023, -.769738477997, -.250000000000, .026595224666, 3.122661756827, .190003957355]
  global u12454u12455u12452u12509u12452u12531u12488_67_q=[-1.9135437459518938, -2.3717387219568336, -1.36633154374372, -1.0932177608774527, 1.5388151300386905, -0.32489438488823286]
  global u12454u12455u12452u12509u12452u12531u12488_68_p=p[-.400000000000, -.769764524263, -.250000000000, .026531939057, 3.122738702253, .190014657192]
  global u12454u12455u12452u12509u12452u12531u12488_68_q=[-1.818862297063192, -2.3106988577225476, -1.483072661381895, -1.039567555772578, 1.5503184080389998, -0.23062355306123106]
  global u12454u12455u12452u12509u12452u12531u12488_69_p=p[-.300000000000, -.769757033912, -.250000000000, .026527276191, 3.122641123221, .190148352440]
  global u12454u12455u12452u12509u12452u12531u12488_69_q=[-1.717697651930628, -2.2633363182227457, -1.5728647610619202, -0.9982571619927505, 1.5628664957611256, -0.12999309911338042]
  global u12454u12455u12452u12509u12452u12531u12488_70_p=p[-.200000000000, -.769859919986, -.250000000000, .026574690387, 3.122642155928, .189875394546]
  global u12454u12455u12452u12509u12452u12531u12488_70_q=[-1.6113376615651154, -2.229116266779524, -1.6374335267785831, -0.9674578160173564, 1.5759949438086123, -0.024246936790873974]
  global u12454u12455u12452u12509u12452u12531u12488_71_p=p[-.100000000000, -.769753066673, -.250000000000, .026570626492, 3.122639670377, .190009590292]
  global u12454u12455u12452u12509u12452u12531u12488_71_q=[-1.501821439881816, -2.2080909569003246, -1.677299501037198, -0.9469871603116431, 1.589307082655564, 0.08456452486400107]
  global u12454u12455u12452u12509u12452u12531u12488_72_p=p[.000000000000, -.769750003345, -.250000000000, .026519903737, 3.122659640697, .189972763518]
  global u12454u12455u12452u12509u12452u12531u12488_72_q=[-1.3916419264178117, -2.2005739153289863, -1.6922310507692249, -0.9363857324454763, 1.602359913212901, 0.19400664438287413]
  global u12454u12455u12452u12509u12452u12531u12488_73_p=p[.100000000000, -.769749556073, -.250000000000, .026619713288, 3.122673196471, .190030383970]
  global u12454u12455u12452u12509u12452u12531u12488_73_q=[-1.2834875706405704, -2.206624931651488, -1.682211080315593, -0.9359177505110488, 1.6147217796817626, 0.3015648852345068]
  global u12454u12455u12452u12509u12452u12531u12488_74_p=p[.200000000000, -.769767367045, -.250000000000, .026579491720, 3.122557456139, .190146936275]
  global u12454u12455u12452u12509u12452u12531u12488_74_q=[-1.1798612316074504, -2.226113812717581, -1.647262133878324, -0.9458966408966809, 1.626129530519922, 0.40457797179985944]
  global u12454u12455u12452u12509u12452u12531u12488_75_p=p[.300000000000, -.769739226409, -.250000000000, .026520993423, 3.122701279074, .190022678776]
  global u12454u12455u12452u12509u12452u12531u12488_75_q=[-1.082420190183452, -2.258611512188663, -1.587640358854391, -0.9667732255880814, 1.635950247287148, 0.5014976807300585]
  global u12454u12455u12452u12509u12452u12531u12488_76_p=p[.400000000000, -.769736890349, -.250000000000, .026578091797, 3.122692098797, .190108965195]
  global u12454u12455u12452u12509u12452u12531u12488_76_q=[-0.9927124676179488, -2.3042197623925653, -1.502581256375688, -0.9996976050411561, 1.644545839530434, 0.5908234016762798]
  global u12454u12455u12452u12509u12452u12531u12488_77_p=p[.500000000000, -.769789067851, -.250000000000, .026451834700, 3.122734551743, .190060963876]
  global u12454u12455u12452u12509u12452u12531u12488_77_q=[-0.911141903906703, -2.363132593354193, -1.3909651845983095, -1.0457729904300983, 1.6516890938375914, 0.6719498708334654]
  global u12454u12455u12452u12509u12452u12531u12488_78_p=p[.500000000000, -.769746259843, -.350000000000, .026632918475, 3.122642546449, .190031917005]
  global u12454u12455u12452u12509u12452u12531u12488_78_q=[-0.911136504370206, -2.4662491161459315, -1.4059144383678088, -0.9276711408227385, 1.6516950704382989, 0.6716132136359318]
  global u12454u12455u12452u12509u12452u12531u12488_79_p=p[.400000000000, -.769754086620, -.350000000000, .026483089559, 3.122665596748, .190070073009]
  global u12454u12455u12452u12509u12452u12531u12488_79_q=[-0.9926947483627249, -2.4130265630898133, -1.5173616574429225, -0.876110033773541, 1.6444562636181184, 0.5903198031027443]
  global u12454u12455u12452u12509u12452u12531u12488_80_p=p[.300000000000, -.769759240242, -.350000000000, .026515155554, 3.122683522897, .189979664284]
  global u12454u12455u12452u12509u12452u12531u12488_80_q=[-1.0824002437921623, -2.372272072567611, -1.602619499340518, -0.8381299029807012, 1.6358258408301474, 0.5010521694080472]
  global u12454u12455u12452u12509u12452u12531u12488_81_p=p[.200000000000, -.769782337339, -.350000000000, .026450672254, 3.122691499402, .190087976014]
  global u12454u12455u12452u12509u12452u12531u12488_81_q=[-1.1797442779124427, -2.3435202232021233, -1.6624820867583336, -0.8133023613201278, 1.6258463189823047, 0.40415578958410325]
  global u12454u12455u12452u12509u12452u12531u12488_82_p=p[.100000000000, -.769770071511, -.350000000000, .026509267542, 3.122615484040, .190166288402]
  global u12454u12455u12452u12509u12452u12531u12488_82_q=[-1.2834909141945703, -2.3264318153944323, -1.697549412973558, -0.8008661515716451, 1.6146194085547307, 0.3010235886202368]
  global u12454u12455u12452u12509u12452u12531u12488_83_p=p[-.000000000000, -.769731783317, -.350000000000, .026501801012, 3.122670299566, .190113607568]
  global u12454u12455u12452u12509u12452u12531u12488_83_q=[-1.3915972123618294, -2.3209839197478868, -1.7078261265448091, -0.800485979493545, 1.6021846725072564, 0.19357754067502775]
  global u12454u12455u12452u12509u12452u12531u12488_84_p=p[-.100000000000, -.769749078146, -.350000000000, .026435540532, 3.122700430020, .190018836303]
  global u12454u12455u12452u12509u12452u12531u12488_84_q=[-1.5017385175061966, -2.3273475655006894, -1.6930568406856494, -0.8119896327077765, 1.589079000749689, 0.08410464727733657]
  global u12454u12455u12452u12509u12452u12531u12488_85_p=p[-.200000000000, -.769742709783, -.350000000000, .026498307507, 3.122661506478, .190063165917]
  global u12454u12455u12452u12509u12452u12531u12488_85_q=[-1.6112832906100572, -2.3455725205239375, -1.6533086926533294, -0.8352472495025722, 1.5758060118940982, -0.024697298817159208]
  global u12454u12455u12452u12509u12452u12531u12488_86_p=p[-.300000000000, -.769789107309, -.350000000000, .026558112637, 3.122633162200, .190053695390]
  global u12454u12455u12452u12509u12452u12531u12488_86_q=[-1.717676826476799, -2.375755707514987, -1.5885678604264202, -0.8700742693097645, 1.562755338205629, -0.13041057498377384]
  global u12454u12455u12452u12509u12452u12531u12488_87_p=p[-.400000000000, -.769750871040, -.350000000000, .026609072555, 3.122576959374, .190130399395]
  global u12454u12455u12452u12509u12452u12531u12488_87_q=[-1.8189161506226643, -2.4180906442553223, -1.4986412069541473, -0.916712545057293, 1.5503386962257162, -0.23108807208201299]
  global u12454u12455u12452u12509u12452u12531u12488_88_p=p[-.500000000000, -.769691340383, -.350000000000, .026559486268, 3.122651936309, .190221807707]
  global u12454u12455u12452u12509u12452u12531u12488_88_q=[-1.913510592416129, -2.4733087206598636, -1.382186318569813, -0.975910801486517, 1.53869884506999, -0.3253309202578123]
  $ 2 "開始前シーケンス"
  $ 6 "ロボットプログラム"
  $ 7 "荷重の設定: k10"
  set_target_payload(0.100000, [0.135000, 0.000000, 0.225000], [10.000000, 10.000000, 10.000000, 0.000000, 0.000000, 0.000000])
  $ 8 "設定"
  set_tcp(p[0.0,0.08,0.42,0.0,0.0,0.0])
  $ 9 "MoveJ"
  $ 10 "gHome_Position" "breakAfter"
  movej(gHome_Position, a=0.17453292519943295, v=0.5235987755982988)
  $ 11 "設定"
  set_tcp(p[0.0,0.08,0.42,1.8940313042642463,0.0,0.0])
  $ 12 "MoveL"
  $ 13 "gGD_1_M_RXF" "breakAfter"
  movel(gGD_1_M_RXF, a=0.05, v=0.15)
  $ 14 "待機: 1.0"
  sleep(1.0)
  $ 15 "gGD_1_LM_RXF" "breakAfter"
  movel(gGD_1_LM_RXF, a=0.05, v=0.15)
  $ 16 "待機: 1.0"
  sleep(1.0)
  $ 17 "gGD_1_RM_RXF" "breakAfter"
  movel(gGD_1_RM_RXF, a=0.05, v=0.15)
  $ 18 "待機: 1.0"
  sleep(1.0)
  $ 19 "gGD_1_M_RXF" "breakAfter"
  movel(gGD_1_M_RXF, a=0.05, v=0.15)
  $ 20 "待機: 1.0"
  sleep(1.0)
  $ 21 "設定"
  set_tcp(p[0.0,0.08,0.42,0.0,0.0,0.0])
  $ 22 "MoveL"
  $ 23 "ウェイポイント_1" "breakAfter"
  movel(u12454u12455u12452u12509u12452u12531u12488_1_p, a=0.05, v=0.15)
  $ 24 "待機: 0.5"
  sleep(0.5)
  $ 25 "ウェイポイント_2" "breakAfter"
  movel(u12454u12455u12452u12509u12452u12531u12488_2_p, a=0.05, v=0.15)
  $ 26 "待機: 0.5"
  sleep(0.5)
  $ 27 "ウェイポイント_3" "breakAfter"
  movel(u12454u12455u12452u12509u12452u12531u12488_3_p, a=0.05, v=0.15)
  $ 28 "待機: 0.5"
  sleep(0.5)
  $ 29 "ウェイポイント_4" "breakAfter"
  movel(u12454u12455u12452u12509u12452u12531u12488_4_p, a=0.05, v=0.15)
  $ 30 "待機: 0.5"
  sleep(0.5)
  $ 31 "ウェイポイント_5" "breakAfter"
  movel(u12454u12455u12452u12509u12452u12531u12488_5_p, a=0.05, v=0.15)
  $ 32 "待機: 0.5"
  sleep(0.5)
  $ 33 "ウェイポイント_6" "breakAfter"
  movel(u12454u12455u12452u12509u12452u12531u12488_6_p, a=0.05, v=0.15)
  $ 34 "待機: 0.5"
  sleep(0.5)
  $ 35 "ウェイポイント_7" "breakAfter"
  movel(u12454u12455u12452u12509u12452u12531u12488_7_p, a=0.05, v=0.15)
  $ 36 "待機: 0.5"
  sleep(0.5)
  $ 37 "ウェイポイント_8" "breakAfter"
  movel(u12454u12455u12452u12509u12452u12531u12488_8_p, a=0.05, v=0.15)
  $ 38 "待機: 0.5"
  sleep(0.5)
  $ 39 "ウェイポイント_9" "breakAfter"
  movel(u12454u12455u12452u12509u12452u12531u12488_9_p, a=0.05, v=0.15)
  $ 40 "待機: 0.5"
  sleep(0.5)
  $ 41 "ウェイポイント_10" "breakAfter"
  movel(u12454u12455u12452u12509u12452u12531u12488_10_p, a=0.05, v=0.15)
  $ 42 "待機: 0.5"
  sleep(0.5)
  $ 43 "ウェイポイント_11" "breakAfter"
  movel(u12454u12455u12452u12509u12452u12531u12488_11_p, a=0.05, v=0.15)
  $ 44 "待機: 0.5"
  sleep(0.5)
  $ 45 "ウェイポイント_12" "breakAfter"
  movel(u12454u12455u12452u12509u12452u12531u12488_12_p, a=0.05, v=0.15)
  $ 46 "待機: 0.5"
  sleep(0.5)
  $ 47 "ウェイポイント_13" "breakAfter"
  movel(u12454u12455u12452u12509u12452u12531u12488_13_p, a=0.05, v=0.15)
  $ 48 "待機: 0.5"
  sleep(0.5)
  $ 49 "ウェイポイント_14" "breakAfter"
  movel(u12454u12455u12452u12509u12452u12531u12488_14_p, a=0.05, v=0.15)
  $ 50 "待機: 0.5"
  sleep(0.5)
  $ 51 "ウェイポイント_15" "breakAfter"
  movel(u12454u12455u12452u12509u12452u12531u12488_15_p, a=0.05, v=0.15)
  $ 52 "待機: 0.5"
  sleep(0.5)
  $ 53 "ウェイポイント_16" "breakAfter"
  movel(u12454u12455u12452u12509u12452u12531u12488_16_p, a=0.05, v=0.15)
  $ 54 "待機: 0.5"
  sleep(0.5)
  $ 55 "ウェイポイント_17" "breakAfter"
  movel(u12454u12455u12452u12509u12452u12531u12488_17_p, a=0.05, v=0.15)
  $ 56 "待機: 0.5"
  sleep(0.5)
  $ 57 "ウェイポイント_18" "breakAfter"
  movel(u12454u12455u12452u12509u12452u12531u12488_18_p, a=0.05, v=0.15)
  $ 58 "待機: 0.5"
  sleep(0.5)
  $ 59 "ウェイポイント_19" "breakAfter"
  movel(u12454u12455u12452u12509u12452u12531u12488_19_p, a=0.05, v=0.15)
  $ 60 "待機: 0.5"
  sleep(0.5)
  $ 61 "ウェイポイント_20" "breakAfter"
  movel(u12454u12455u12452u12509u12452u12531u12488_20_p, a=0.05, v=0.15)
  $ 62 "待機: 0.5"
  sleep(0.5)
  $ 63 "ウェイポイント_21" "breakAfter"
  movel(u12454u12455u12452u12509u12452u12531u12488_21_p, a=0.05, v=0.15)
  $ 64 "待機: 0.5"
  sleep(0.5)
  $ 65 "ウェイポイント_22" "breakAfter"
  movel(u12454u12455u12452u12509u12452u12531u12488_22_p, a=0.05, v=0.15)
  $ 66 "待機: 0.5"
  sleep(0.5)
  $ 67 "ウェイポイント_23" "breakAfter"
  movel(u12454u12455u12452u12509u12452u12531u12488_23_p, a=0.05, v=0.15)
  $ 68 "待機: 0.5"
  sleep(0.5)
  $ 69 "ウェイポイント_24" "breakAfter"
  movel(u12454u12455u12452u12509u12452u12531u12488_24_p, a=0.05, v=0.15)
  $ 70 "待機: 0.5"
  sleep(0.5)
  $ 71 "ウェイポイント_25" "breakAfter"
  movel(u12454u12455u12452u12509u12452u12531u12488_25_p, a=0.05, v=0.15)
  $ 72 "待機: 0.5"
  sleep(0.5)
  $ 73 "ウェイポイント_26" "breakAfter"
  movel(u12454u12455u12452u12509u12452u12531u12488_26_p, a=0.05, v=0.15)
  $ 74 "待機: 0.5"
  sleep(0.5)
  $ 75 "ウェイポイント_27" "breakAfter"
  movel(u12454u12455u12452u12509u12452u12531u12488_27_p, a=0.05, v=0.15)
  $ 76 "待機: 0.5"
  sleep(0.5)
  $ 77 "ウェイポイント_28" "breakAfter"
  movel(u12454u12455u12452u12509u12452u12531u12488_28_p, a=0.05, v=0.15)
  $ 78 "待機: 0.5"
  sleep(0.5)
  $ 79 "ウェイポイント_29" "breakAfter"
  movel(u12454u12455u12452u12509u12452u12531u12488_29_p, a=0.05, v=0.15)
  $ 80 "待機: 0.5"
  sleep(0.5)
  $ 81 "ウェイポイント_30" "breakAfter"
  movel(u12454u12455u12452u12509u12452u12531u12488_30_p, a=0.05, v=0.15)
  $ 82 "待機: 0.5"
  sleep(0.5)
  $ 83 "ウェイポイント_31" "breakAfter"
  movel(u12454u12455u12452u12509u12452u12531u12488_31_p, a=0.05, v=0.15)
  $ 84 "待機: 0.5"
  sleep(0.5)
  $ 85 "ウェイポイント_32" "breakAfter"
  movel(u12454u12455u12452u12509u12452u12531u12488_32_p, a=0.05, v=0.15)
  $ 86 "待機: 0.5"
  sleep(0.5)
  $ 87 "ウェイポイント_33" "breakAfter"
  movel(u12454u12455u12452u12509u12452u12531u12488_33_p, a=0.05, v=0.15)
  $ 88 "待機: 0.5"
  sleep(0.5)
  $ 89 "ウェイポイント_34" "breakAfter"
  movel(u12454u12455u12452u12509u12452u12531u12488_34_p, a=0.05, v=0.15)
  $ 90 "待機: 0.5"
  sleep(0.5)
  $ 91 "ウェイポイント_35" "breakAfter"
  movel(u12454u12455u12452u12509u12452u12531u12488_35_p, a=0.05, v=0.15)
  $ 92 "待機: 0.5"
  sleep(0.5)
  $ 93 "ウェイポイント_36" "breakAfter"
  movel(u12454u12455u12452u12509u12452u12531u12488_36_p, a=0.05, v=0.15)
  $ 94 "待機: 0.5"
  sleep(0.5)
  $ 95 "ウェイポイント_37" "breakAfter"
  movel(u12454u12455u12452u12509u12452u12531u12488_37_p, a=0.05, v=0.15)
  $ 96 "待機: 0.5"
  sleep(0.5)
  $ 97 "ウェイポイント_38" "breakAfter"
  movel(u12454u12455u12452u12509u12452u12531u12488_38_p, a=0.05, v=0.15)
  $ 98 "待機: 0.5"
  sleep(0.5)
  $ 99 "ウェイポイント_39" "breakAfter"
  movel(u12454u12455u12452u12509u12452u12531u12488_39_p, a=0.05, v=0.15)
  $ 100 "待機: 0.5"
  sleep(0.5)
  $ 101 "ウェイポイント_40" "breakAfter"
  movel(u12454u12455u12452u12509u12452u12531u12488_40_p, a=0.05, v=0.15)
  $ 102 "待機: 0.5"
  sleep(0.5)
  $ 103 "ウェイポイント_41" "breakAfter"
  movel(u12454u12455u12452u12509u12452u12531u12488_41_p, a=0.05, v=0.15)
  $ 104 "待機: 0.5"
  sleep(0.5)
  $ 105 "ウェイポイント_42" "breakAfter"
  movel(u12454u12455u12452u12509u12452u12531u12488_42_p, a=0.05, v=0.15)
  $ 106 "待機: 0.5"
  sleep(0.5)
  $ 107 "ウェイポイント_43" "breakAfter"
  movel(u12454u12455u12452u12509u12452u12531u12488_43_p, a=0.05, v=0.15)
  $ 108 "待機: 0.5"
  sleep(0.5)
  $ 109 "ウェイポイント_44" "breakAfter"
  movel(u12454u12455u12452u12509u12452u12531u12488_44_p, a=0.05, v=0.15)
  $ 110 "待機: 0.5"
  sleep(0.5)
  $ 111 "ウェイポイント_45" "breakAfter"
  movel(u12454u12455u12452u12509u12452u12531u12488_45_p, a=0.05, v=0.15)
  $ 112 "待機: 0.5"
  sleep(0.5)
  $ 113 "ウェイポイント_46" "breakAfter"
  movel(u12454u12455u12452u12509u12452u12531u12488_46_p, a=0.05, v=0.15)
  $ 114 "待機: 0.5"
  sleep(0.5)
  $ 115 "ウェイポイント_47" "breakAfter"
  movel(u12454u12455u12452u12509u12452u12531u12488_47_p, a=0.05, v=0.15)
  $ 116 "待機: 0.5"
  sleep(0.5)
  $ 117 "ウェイポイント_48" "breakAfter"
  movel(u12454u12455u12452u12509u12452u12531u12488_48_p, a=0.05, v=0.15)
  $ 118 "待機: 0.5"
  sleep(0.5)
  $ 119 "ウェイポイント_49" "breakAfter"
  movel(u12454u12455u12452u12509u12452u12531u12488_49_p, a=0.05, v=0.15)
  $ 120 "待機: 0.5"
  sleep(0.5)
  $ 121 "ウェイポイント_50" "breakAfter"
  movel(u12454u12455u12452u12509u12452u12531u12488_50_p, a=0.05, v=0.15)
  $ 122 "待機: 0.5"
  sleep(0.5)
  $ 123 "ウェイポイント_51" "breakAfter"
  movel(u12454u12455u12452u12509u12452u12531u12488_51_p, a=0.05, v=0.15)
  $ 124 "待機: 0.5"
  sleep(0.5)
  $ 125 "ウェイポイント_52" "breakAfter"
  movel(u12454u12455u12452u12509u12452u12531u12488_52_p, a=0.05, v=0.15)
  $ 126 "待機: 0.5"
  sleep(0.5)
  $ 127 "ウェイポイント_53" "breakAfter"
  movel(u12454u12455u12452u12509u12452u12531u12488_53_p, a=0.05, v=0.15)
  $ 128 "待機: 0.5"
  sleep(0.5)
  $ 129 "ウェイポイント_54" "breakAfter"
  movel(u12454u12455u12452u12509u12452u12531u12488_54_p, a=0.05, v=0.15)
  $ 130 "待機: 0.5"
  sleep(0.5)
  $ 131 "ウェイポイント_55" "breakAfter"
  movel(u12454u12455u12452u12509u12452u12531u12488_55_p, a=0.05, v=0.15)
  $ 132 "待機: 0.5"
  sleep(0.5)
  $ 133 "ウェイポイント_56" "breakAfter"
  movel(u12454u12455u12452u12509u12452u12531u12488_56_p, a=0.05, v=0.15)
  $ 134 "待機: 0.5"
  sleep(0.5)
  $ 135 "ウェイポイント_57" "breakAfter"
  movel(u12454u12455u12452u12509u12452u12531u12488_57_p, a=0.05, v=0.15)
  $ 136 "待機: 0.5"
  sleep(0.5)
  $ 137 "ウェイポイント_58" "breakAfter"
  movel(u12454u12455u12452u12509u12452u12531u12488_58_p, a=0.05, v=0.15)
  $ 138 "待機: 0.5"
  sleep(0.5)
  $ 139 "ウェイポイント_59" "breakAfter"
  movel(u12454u12455u12452u12509u12452u12531u12488_59_p, a=0.05, v=0.15)
  $ 140 "待機: 0.5"
  sleep(0.5)
  $ 141 "ウェイポイント_60" "breakAfter"
  movel(u12454u12455u12452u12509u12452u12531u12488_60_p, a=0.05, v=0.15)
  $ 142 "待機: 0.5"
  sleep(0.5)
  $ 143 "ウェイポイント_61" "breakAfter"
  movel(u12454u12455u12452u12509u12452u12531u12488_61_p, a=0.05, v=0.15)
  $ 144 "待機: 0.5"
  sleep(0.5)
  $ 145 "ウェイポイント_62" "breakAfter"
  movel(u12454u12455u12452u12509u12452u12531u12488_62_p, a=0.05, v=0.15)
  $ 146 "待機: 0.5"
  sleep(0.5)
  $ 147 "ウェイポイント_63" "breakAfter"
  movel(u12454u12455u12452u12509u12452u12531u12488_63_p, a=0.05, v=0.15)
  $ 148 "待機: 0.5"
  sleep(0.5)
  $ 149 "ウェイポイント_64" "breakAfter"
  movel(u12454u12455u12452u12509u12452u12531u12488_64_p, a=0.05, v=0.15)
  $ 150 "待機: 0.5"
  sleep(0.5)
  $ 151 "ウェイポイント_65" "breakAfter"
  movel(u12454u12455u12452u12509u12452u12531u12488_65_p, a=0.05, v=0.15)
  $ 152 "待機: 0.5"
  sleep(0.5)
  $ 153 "ウェイポイント_66" "breakAfter"
  movel(u12454u12455u12452u12509u12452u12531u12488_66_p, a=0.05, v=0.15)
  $ 154 "待機: 0.5"
  sleep(0.5)
  $ 155 "ウェイポイント_67" "breakAfter"
  movel(u12454u12455u12452u12509u12452u12531u12488_67_p, a=0.05, v=0.15)
  $ 156 "待機: 0.5"
  sleep(0.5)
  $ 157 "ウェイポイント_68" "breakAfter"
  movel(u12454u12455u12452u12509u12452u12531u12488_68_p, a=0.05, v=0.15)
  $ 158 "待機: 0.5"
  sleep(0.5)
  $ 159 "ウェイポイント_69" "breakAfter"
  movel(u12454u12455u12452u12509u12452u12531u12488_69_p, a=0.05, v=0.15)
  $ 160 "待機: 0.5"
  sleep(0.5)
  $ 161 "ウェイポイント_70" "breakAfter"
  movel(u12454u12455u12452u12509u12452u12531u12488_70_p, a=0.05, v=0.15)
  $ 162 "待機: 0.5"
  sleep(0.5)
  $ 163 "ウェイポイント_71" "breakAfter"
  movel(u12454u12455u12452u12509u12452u12531u12488_71_p, a=0.05, v=0.15)
  $ 164 "待機: 0.5"
  sleep(0.5)
  $ 165 "ウェイポイント_72" "breakAfter"
  movel(u12454u12455u12452u12509u12452u12531u12488_72_p, a=0.05, v=0.15)
  $ 166 "待機: 0.5"
  sleep(0.5)
  $ 167 "ウェイポイント_73" "breakAfter"
  movel(u12454u12455u12452u12509u12452u12531u12488_73_p, a=0.05, v=0.15)
  $ 168 "待機: 0.5"
  sleep(0.5)
  $ 169 "ウェイポイント_74" "breakAfter"
  movel(u12454u12455u12452u12509u12452u12531u12488_74_p, a=0.05, v=0.15)
  $ 170 "待機: 0.5"
  sleep(0.5)
  $ 171 "ウェイポイント_75" "breakAfter"
  movel(u12454u12455u12452u12509u12452u12531u12488_75_p, a=0.05, v=0.15)
  $ 172 "待機: 0.5"
  sleep(0.5)
  $ 173 "ウェイポイント_76" "breakAfter"
  movel(u12454u12455u12452u12509u12452u12531u12488_76_p, a=0.05, v=0.15)
  $ 174 "待機: 0.5"
  sleep(0.5)
  $ 175 "ウェイポイント_77" "breakAfter"
  movel(u12454u12455u12452u12509u12452u12531u12488_77_p, a=0.05, v=0.15)
  $ 176 "待機: 0.5"
  sleep(0.5)
  $ 177 "ウェイポイント_78" "breakAfter"
  movel(u12454u12455u12452u12509u12452u12531u12488_78_p, a=0.05, v=0.15)
  $ 178 "待機: 0.5"
  sleep(0.5)
  $ 179 "ウェイポイント_79" "breakAfter"
  movel(u12454u12455u12452u12509u12452u12531u12488_79_p, a=0.05, v=0.15)
  $ 180 "待機: 0.5"
  sleep(0.5)
  $ 181 "ウェイポイント_80" "breakAfter"
  movel(u12454u12455u12452u12509u12452u12531u12488_80_p, a=0.05, v=0.15)
  $ 182 "待機: 0.5"
  sleep(0.5)
  $ 183 "ウェイポイント_81" "breakAfter"
  movel(u12454u12455u12452u12509u12452u12531u12488_81_p, a=0.05, v=0.15)
  $ 184 "待機: 0.5"
  sleep(0.5)
  $ 185 "ウェイポイント_82" "breakAfter"
  movel(u12454u12455u12452u12509u12452u12531u12488_82_p, a=0.05, v=0.15)
  $ 186 "待機: 0.5"
  sleep(0.5)
  $ 187 "ウェイポイント_83" "breakAfter"
  movel(u12454u12455u12452u12509u12452u12531u12488_83_p, a=0.05, v=0.15)
  $ 188 "待機: 0.5"
  sleep(0.5)
  $ 189 "ウェイポイント_84" "breakAfter"
  movel(u12454u12455u12452u12509u12452u12531u12488_84_p, a=0.05, v=0.15)
  $ 190 "待機: 0.5"
  sleep(0.5)
  $ 191 "ウェイポイント_85" "breakAfter"
  movel(u12454u12455u12452u12509u12452u12531u12488_85_p, a=0.05, v=0.15)
  $ 192 "待機: 0.5"
  sleep(0.5)
  $ 193 "ウェイポイント_86" "breakAfter"
  movel(u12454u12455u12452u12509u12452u12531u12488_86_p, a=0.05, v=0.15)
  $ 194 "待機: 0.5"
  sleep(0.5)
  $ 195 "ウェイポイント_87" "breakAfter"
  movel(u12454u12455u12452u12509u12452u12531u12488_87_p, a=0.05, v=0.15)
  $ 196 "待機: 0.5"
  sleep(0.5)
  $ 197 "ウェイポイント_88" "breakAfter"
  movel(u12454u12455u12452u12509u12452u12531u12488_88_p, a=0.05, v=0.15)
  $ 198 "待機: 0.5"
  sleep(0.5)
  $ 199 "MoveJ"
  $ 200 "gHome_Position" "breakAfter"
  movej(gHome_Position, a=0.17453292519943295, v=0.5235987755982988)
  $ 201 "停止"
  halt
end
